FUNCTION_BLOCK FB_Room IMPLEMENTS  I_Room
VAR_INPUT
END_VAR
VAR_OUTPUT
END_VAR
VAR
END_VAR

{warning 'add method implementation'}
(* sets the temperature, returns the actual status*)
METHOD M_SetTemperature : BOOL
VAR_INPUT
	bOnOff	: BOOL;
	nTemperature	: REAL;
END_VAR
END_METHOD

{warning 'add method implementation'}
(* Switches the light on/off with certain illuminance*)
METHOD M_SwitchLight : BOOL
VAR_INPUT
	bOnOff	: BOOL;
	nIlluminance	: REAL;
END_VAR
END_METHOD

END_FUNCTION_BLOCK

(* stored: Version 1.1.0.1, ProductVersion 3.1.4022.18
   POU FB_Room: Id {eb5ffc53-f4dc-4c58-ac7d-796ce77112a6}, SpecialFunc None
   Method M_SetTemperature: Id {4a8201b3-3769-45e8-a8d3-3fd5d308d43d}
   Method M_SwitchLight: Id {6d5fde6e-9d37-4a59-9f5b-20302e203c89} *)
